// TwinCAT 3 PLC project Motor_test
// ProgramVersion: 3.1.4023.0
// libraries:
//   Tc2_ControllerToolbox, * (Beckhoff Automation GmbH)
//   Tc2_MC2, * (Beckhoff Automation GmbH)
//   Tc2_NCI, * (Beckhoff Automation GmbH)
//   Tc2_NcKinematicTransformation, * (Beckhoff Automation GmbH)
//   Tc2_PlcInterpolation, * (Beckhoff Automation GmbH)
//   Tc2_Standard, * (Beckhoff Automation GmbH)
//   Tc2_System, * (Beckhoff Automation GmbH)
//   Tc3_Module, * (Beckhoff Automation GmbH)
//   VisuSymbols,3.5.10.0,System
// project tree:
//   / GlobalTextList.TcGTLO, PlcTask.TcTTO, Visualization Manager.TcVMO (not stored)
//   POUs/ FB_CheckCurrentState.TcPOU, FB_ExecuteGcode.TcPOU, FB_GetPrinterParameters.TcPOU, FB_GetTemperature.TcPOU, FB_PowerChannel.TcPOU, FB_SteinhartEquation.TcPOU, Heater_control.TcPOU, MAIN.TcPOU, FB_PWM.TcPOU
//   VISUs/ Visualization.TcVIS
// real-time tasks:
//   TASK PlcTask: cycle T#1ms, priority 20, ADS port 350
// motion (NC):
//   TASK NC-Task 1 SAF: cycle T#1ms, priority 4, ADS port 501
//   TASK NC-Task 1 SVB: cycle T#1ms, priority 8, ADS port 511
//   AXIS axis xy 1 (id 1)
//     Dynamic: AccelerationMaximum=2000, DecelerationMaximum=2000, Acceleration=1000, Deceleration=1000
//     Velo: SlowManual=50, FastManual=100, Maximum=500
//     OtherSettings: AllowMotionCmdToSlave=true
//     encoder EncType=4
//       EncPara: ScaleFactorNumerator=40, ScaleFactorDenominator=12800, MaxCount=#x0000ffff
//         Inc: RefSoftSyncMask=#x0000ffff
//     drive DrvType=24
//       Analog: VeloReferenz=400, TorqueSetpointScale=10, ScaleFactorActTorque=0.1
//       TimeComp: TaskDelayCycles=1
//     controller CtrType=1
//       CtrPara: PriorControlFactor=1
//         Observer: BandWidth=20
//   AXIS axis xy 2 (id 2)
//     Dynamic: AccelerationMaximum=2000, DecelerationMaximum=2000, Acceleration=1000, Deceleration=1000
//     Velo: SlowManual=50, FastManual=100, Maximum=500
//     OtherSettings: AllowMotionCmdToSlave=true
//     encoder EncType=4
//       EncPara: ScaleFactorNumerator=40, ScaleFactorDenominator=12800, MaxCount=#x0000ffff
//         Inc: RefSoftSyncMask=#x0000ffff
//     drive DrvType=24
//       Analog: VeloReferenz=400, TorqueSetpointScale=10, ScaleFactorActTorque=0.1
//       TimeComp: TaskDelayCycles=1
//     controller CtrType=1
//       CtrPara: PriorControlFactor=1
//         Observer: BandWidth=20
//   AXIS Z axis (id 3)
//     Dynamic: AccelerationMaximum=100, DecelerationMaximum=100, Acceleration=50, Deceleration=50, Jerk=1000
//     Velo: RefSearch=3, RefSync=3, SlowManual=1, FastManual=4, Maximum=10
//     OtherSettings: AllowMotionCmdToSlave=true
//     encoder EncType=4
//       EncPara: ScaleFactorNumerator=8, ScaleFactorDenominator=12800, MaxCount=#x0000ffff
//         SoftEndMaxControl: Range=400
//         Inc: RefSearchInverse=true, RefSyncInverse=false, RefPosition=0.4, RefMode=1, RefSoftSyncMask=#x0000ffff
//     drive DrvType=24
//       Analog: VeloReferenz=80, TorqueSetpointScale=10, ScaleFactorActTorque=0.1
//       TimeComp: TaskDelayCycles=1
//     controller CtrType=1
//       CtrPara: PriorControlFactor=1
//         Observer: BandWidth=20
//   AXIS Extruder (id 4)
//     Dynamic: AccelerationMaximum=400, DecelerationMaximum=400, Acceleration=200, Deceleration=200, Jerk=500
//     Velo: SlowManual=1, FastManual=2, Maximum=100
//     OtherSettings: AllowMotionCmdToSlave=true
//     encoder EncType=4
//       EncPara: ScaleFactorNumerator=22.857, ScaleFactorDenominator=12800, MaxCount=#x0000ffff
//         Inc: RefSoftSyncMask=#x0000ffff
//     drive DrvType=24
//       Analog: VeloReferenz=50, TorqueSetpointScale=10, ScaleFactorActTorque=0.1
//       TimeComp: TaskDelayCycles=1
//     controller CtrType=1
//       CtrPara: PriorControlFactor=1
//         PosDiffControl: Range=15
//         Observer: BandWidth=20
//   AXIS X axis (id 5)
//     Dynamic: AccelerationMaximum=2000, DecelerationMaximum=2000, Acceleration=1000, Deceleration=1000
//     Velo: RefSearch=20, RefSync=20, SlowManual=20, FastManual=40, Maximum=500
//     OtherSettings: AllowMotionCmdToSlave=true
//     encoder EncType=1
//       EncPara: ScaleFactorNumerator=1, ScaleFactorDenominator=0.1
//         SoftEndMaxControl: Range=300
//     drive DrvType=5
//       Analog: VeloReferenz=500, TorqueSetpointScale=10, ScaleFactorActTorque=0.1
//       TimeComp: TaskDelayCycles=1
//     controller CtrType=1
//       CtrPara: PriorControlFactor=1
//         Observer: BandWidth=20
//   AXIS Y axis (id 6)
//     Dynamic: AccelerationMaximum=2000, DecelerationMaximum=2000, Acceleration=1000, Deceleration=1000
//     Velo: RefSearch=15, RefSync=15, SlowManual=15, FastManual=40, Maximum=500
//     OtherSettings: AllowMotionCmdToSlave=true
//     encoder EncType=1
//       SoftEndMaxControl: Range=300
//     drive DrvType=5
//       Analog: VeloReferenz=500, TorqueSetpointScale=10, ScaleFactorActTorque=0.1
//       TimeComp: TaskDelayCycles=1
//     controller CtrType=1
//       CtrPara: PriorControlFactor=1
//         Observer: BandWidth=20
// I/O:
//   DEVICE Device 3 (EtherCAT), AmsNetId 5.68.190.166.4.1
//     Term 1 (EK1101) [EK1101 EtherCAT Coupler (2A E-Bus, ID switch)]
//       Term 2 (EL9227-5500) [EL9227-5500 Overcurrent protection 24V DC, 2Ch., max. 10A (sum), adjustable, extended functionalities]
//       Term 3 (EL2024) [EL2024 4Ch. Dig. Output 24V, 2A]
//       Term 15 (EL3204-0200) [EL3204-0200 4Ch. Ana. In. PT1000 (RTD)]
//       Term 5 (EL1004) [EL1004 4Ch. Dig. Input 24V, 3ms]
//       Term 6 (EL7037) [EL7037 1Ch. Stepper motor output stage (24V, 1.5A)]
//       Term 7 (EL7037) [EL7037 1Ch. Stepper motor output stage (24V, 1.5A)]
//       Term 8 (EL7037) [EL7037 1Ch. Stepper motor output stage (24V, 1.5A)]
//       Term 9 (EL7037) [EL7037 1Ch. Stepper motor output stage (24V, 1.5A)]
//       Term 10 (EL9227-5500) [EL9227-5500 Overcurrent protection 24V DC, 2Ch., max. 10A (sum), adjustable, extended functionalities]
//       Term 11 (EL9011) [EL9011 End Terminal]
// variable links:
//   NC-Task 1 SAF/Axes/Extruder <-> Device 3 (EtherCAT)/Term 1 (EK1101)/Term 9 (EL7037)
//     Drive/Inputs/In/nState1 @bit 3 <-> STM Status/Status/Error
//     Drive/Inputs/In/nState1 @bit 7 <-> STM Status/Status/Motor stall
//     Drive/Inputs/In/nState1 @bit 5 <-> STM Status/Status/Moving negative
//     Drive/Inputs/In/nState1 @bit 4 <-> STM Status/Status/Moving positive
//     Drive/Inputs/In/nState1 @bit 1 <-> STM Status/Status/Ready
//     Drive/Inputs/In/nState1 <-> STM Status/Status/Ready to enable
//     Drive/Inputs/In/nState1 @bit 6 <-> STM Status/Status/Torque reduced
//     Drive/Inputs/In/nState1 @bit 2 <-> STM Status/Status/Warning
//     Drive/Inputs/In/nState2 @bit 3 <-> STM Status/Status/Digital input 1
//     Drive/Inputs/In/nState2 @bit 4 <-> STM Status/Status/Digital input 2
//     Drive/Inputs/In/nState2 @bit 5 <-> STM Status/Status/Sync error
//     Drive/Inputs/In/nState2 @bit 7 <-> STM Status/Status/TxPDO Toggle
//     Drive/Inputs/In/nState4 @bit 1 <-> WcState/InputToggle
//     Drive/Inputs/In/nState4 <-> WcState/WcState
//     Drive/Outputs/Out/nCtrl1 <-> STM Control/Control/Enable
//     Drive/Outputs/Out/nCtrl1 @bit 2 <-> STM Control/Control/Reduce torque
//     Drive/Outputs/Out/nCtrl1 @bit 1 <-> STM Control/Control/Reset
//     Drive/Outputs/Out/nCtrl2 @bit 3 <-> STM Control/Control/Digital output 1
//     Drive/Outputs/Out/nDataOut2[0] <-> STM Velocity/Velocity
//     Enc/Inputs/In/nDataIn1[0] <-> ENC Status compact/Counter value
//     Enc/Inputs/In/nDataIn2[0] <-> ENC Status compact/Latch value
//     Enc/Inputs/In/nState1 @bit 4 <-> ENC Status compact/Status/Counter overflow
//     Enc/Inputs/In/nState1 @bit 3 <-> ENC Status compact/Status/Counter underflow
//     Enc/Inputs/In/nState1 @bit 7 <-> ENC Status compact/Status/Extrapolation stall
//     Enc/Inputs/In/nState1 <-> ENC Status compact/Status/Latch C valid
//     Enc/Inputs/In/nState1 @bit 1 <-> ENC Status compact/Status/Latch extern valid
//     Enc/Inputs/In/nState1 @bit 2 <-> ENC Status compact/Status/Set counter done
//     Enc/Inputs/In/nState2 @bit 4 <-> ENC Status compact/Status/Status of extern latch
//     Enc/Inputs/In/nState2 <-> ENC Status compact/Status/Status of input A
//     Enc/Inputs/In/nState2 @bit 1 <-> ENC Status compact/Status/Status of input B
//     Enc/Inputs/In/nState2 @bit 2 <-> ENC Status compact/Status/Status of input C
//     Enc/Inputs/In/nState2 @bit 5 <-> ENC Status compact/Status/Sync error
//     Enc/Inputs/In/nState2 @bit 7 <-> ENC Status compact/Status/TxPDO Toggle
//     Enc/Inputs/In/nState4 @bit 1 <-> WcState/InputToggle
//     Enc/Inputs/In/nState4 <-> WcState/WcState
//     Enc/Outputs/Out/nCtrl1 <-> ENC Control compact/Control/Enable latch C
//     Enc/Outputs/Out/nCtrl1 @bit 3 <-> ENC Control compact/Control/Enable latch extern on negative edge
//     Enc/Outputs/Out/nCtrl1 @bit 1 <-> ENC Control compact/Control/Enable latch extern on positive edge
//     Enc/Outputs/Out/nCtrl1 @bit 2 <-> ENC Control compact/Control/Set counter
//     Enc/Outputs/Out/nDataOut1[0] <-> ENC Control compact/Set counter value
//   NC-Task 1 SAF/Axes/Z axis <-> Device 3 (EtherCAT)/Term 1 (EK1101)/Term 8 (EL7037)
//     Drive/Inputs/In/nState1 @bit 3 <-> STM Status/Status/Error
//     Drive/Inputs/In/nState1 @bit 7 <-> STM Status/Status/Motor stall
//     Drive/Inputs/In/nState1 @bit 5 <-> STM Status/Status/Moving negative
//     Drive/Inputs/In/nState1 @bit 4 <-> STM Status/Status/Moving positive
//     Drive/Inputs/In/nState1 @bit 1 <-> STM Status/Status/Ready
//     Drive/Inputs/In/nState1 <-> STM Status/Status/Ready to enable
//     Drive/Inputs/In/nState1 @bit 6 <-> STM Status/Status/Torque reduced
//     Drive/Inputs/In/nState1 @bit 2 <-> STM Status/Status/Warning
//     Drive/Inputs/In/nState2 @bit 3 <-> STM Status/Status/Digital input 1
//     Drive/Inputs/In/nState2 @bit 4 <-> STM Status/Status/Digital input 2
//     Drive/Inputs/In/nState2 @bit 5 <-> STM Status/Status/Sync error
//     Drive/Inputs/In/nState2 @bit 7 <-> STM Status/Status/TxPDO Toggle
//     Drive/Inputs/In/nState4 @bit 1 <-> WcState/InputToggle
//     Drive/Inputs/In/nState4 <-> WcState/WcState
//     Drive/Outputs/Out/nCtrl1 <-> STM Control/Control/Enable
//     Drive/Outputs/Out/nCtrl1 @bit 2 <-> STM Control/Control/Reduce torque
//     Drive/Outputs/Out/nCtrl1 @bit 1 <-> STM Control/Control/Reset
//     Drive/Outputs/Out/nCtrl2 @bit 3 <-> STM Control/Control/Digital output 1
//     Drive/Outputs/Out/nDataOut2[0] <-> STM Velocity/Velocity
//     Enc/Inputs/In/nDataIn1[0] <-> ENC Status compact/Counter value
//     Enc/Inputs/In/nDataIn2[0] <-> ENC Status compact/Latch value
//     Enc/Inputs/In/nState1 @bit 4 <-> ENC Status compact/Status/Counter overflow
//     Enc/Inputs/In/nState1 @bit 3 <-> ENC Status compact/Status/Counter underflow
//     Enc/Inputs/In/nState1 @bit 7 <-> ENC Status compact/Status/Extrapolation stall
//     Enc/Inputs/In/nState1 <-> ENC Status compact/Status/Latch C valid
//     Enc/Inputs/In/nState1 @bit 1 <-> ENC Status compact/Status/Latch extern valid
//     Enc/Inputs/In/nState1 @bit 2 <-> ENC Status compact/Status/Set counter done
//     Enc/Inputs/In/nState2 @bit 4 <-> ENC Status compact/Status/Status of extern latch
//     Enc/Inputs/In/nState2 <-> ENC Status compact/Status/Status of input A
//     Enc/Inputs/In/nState2 @bit 1 <-> ENC Status compact/Status/Status of input B
//     Enc/Inputs/In/nState2 @bit 2 <-> ENC Status compact/Status/Status of input C
//     Enc/Inputs/In/nState2 @bit 5 <-> ENC Status compact/Status/Sync error
//     Enc/Inputs/In/nState2 @bit 7 <-> ENC Status compact/Status/TxPDO Toggle
//     Enc/Inputs/In/nState4 @bit 1 <-> WcState/InputToggle
//     Enc/Inputs/In/nState4 <-> WcState/WcState
//     Enc/Outputs/Out/nCtrl1 <-> ENC Control compact/Control/Enable latch C
//     Enc/Outputs/Out/nCtrl1 @bit 3 <-> ENC Control compact/Control/Enable latch extern on negative edge
//     Enc/Outputs/Out/nCtrl1 @bit 1 <-> ENC Control compact/Control/Enable latch extern on positive edge
//     Enc/Outputs/Out/nCtrl1 @bit 2 <-> ENC Control compact/Control/Set counter
//     Enc/Outputs/Out/nDataOut1[0] <-> ENC Control compact/Set counter value
//   NC-Task 1 SAF/Axes/axis xy 1 <-> Device 3 (EtherCAT)/Term 1 (EK1101)/Term 6 (EL7037)
//     Drive/Inputs/In/nState1 @bit 3 <-> STM Status/Status/Error
//     Drive/Inputs/In/nState1 @bit 7 <-> STM Status/Status/Motor stall
//     Drive/Inputs/In/nState1 @bit 5 <-> STM Status/Status/Moving negative
//     Drive/Inputs/In/nState1 @bit 4 <-> STM Status/Status/Moving positive
//     Drive/Inputs/In/nState1 @bit 1 <-> STM Status/Status/Ready
//     Drive/Inputs/In/nState1 <-> STM Status/Status/Ready to enable
//     Drive/Inputs/In/nState1 @bit 6 <-> STM Status/Status/Torque reduced
//     Drive/Inputs/In/nState1 @bit 2 <-> STM Status/Status/Warning
//     Drive/Inputs/In/nState2 @bit 3 <-> STM Status/Status/Digital input 1
//     Drive/Inputs/In/nState2 @bit 4 <-> STM Status/Status/Digital input 2
//     Drive/Inputs/In/nState2 @bit 5 <-> STM Status/Status/Sync error
//     Drive/Inputs/In/nState2 @bit 7 <-> STM Status/Status/TxPDO Toggle
//     Drive/Inputs/In/nState4 @bit 1 <-> WcState/InputToggle
//     Drive/Inputs/In/nState4 <-> WcState/WcState
//     Drive/Outputs/Out/nCtrl1 <-> STM Control/Control/Enable
//     Drive/Outputs/Out/nCtrl1 @bit 2 <-> STM Control/Control/Reduce torque
//     Drive/Outputs/Out/nCtrl1 @bit 1 <-> STM Control/Control/Reset
//     Drive/Outputs/Out/nCtrl2 @bit 3 <-> STM Control/Control/Digital output 1
//     Drive/Outputs/Out/nDataOut2[0] <-> STM Velocity/Velocity
//     Enc/Inputs/In/nDataIn1[0] <-> ENC Status compact/Counter value
//     Enc/Inputs/In/nDataIn2[0] <-> ENC Status compact/Latch value
//     Enc/Inputs/In/nState1 @bit 4 <-> ENC Status compact/Status/Counter overflow
//     Enc/Inputs/In/nState1 @bit 3 <-> ENC Status compact/Status/Counter underflow
//     Enc/Inputs/In/nState1 @bit 7 <-> ENC Status compact/Status/Extrapolation stall
//     Enc/Inputs/In/nState1 <-> ENC Status compact/Status/Latch C valid
//     Enc/Inputs/In/nState1 @bit 1 <-> ENC Status compact/Status/Latch extern valid
//     Enc/Inputs/In/nState1 @bit 2 <-> ENC Status compact/Status/Set counter done
//     Enc/Inputs/In/nState2 @bit 4 <-> ENC Status compact/Status/Status of extern latch
//     Enc/Inputs/In/nState2 <-> ENC Status compact/Status/Status of input A
//     Enc/Inputs/In/nState2 @bit 1 <-> ENC Status compact/Status/Status of input B
//     Enc/Inputs/In/nState2 @bit 2 <-> ENC Status compact/Status/Status of input C
//     Enc/Inputs/In/nState2 @bit 5 <-> ENC Status compact/Status/Sync error
//     Enc/Inputs/In/nState2 @bit 7 <-> ENC Status compact/Status/TxPDO Toggle
//     Enc/Inputs/In/nState4 @bit 1 <-> WcState/InputToggle
//     Enc/Inputs/In/nState4 <-> WcState/WcState
//     Enc/Outputs/Out/nCtrl1 <-> ENC Control compact/Control/Enable latch C
//     Enc/Outputs/Out/nCtrl1 @bit 3 <-> ENC Control compact/Control/Enable latch extern on negative edge
//     Enc/Outputs/Out/nCtrl1 @bit 1 <-> ENC Control compact/Control/Enable latch extern on positive edge
//     Enc/Outputs/Out/nCtrl1 @bit 2 <-> ENC Control compact/Control/Set counter
//     Enc/Outputs/Out/nDataOut1[0] <-> ENC Control compact/Set counter value
//   NC-Task 1 SAF/Axes/axis xy 2 <-> Device 3 (EtherCAT)/Term 1 (EK1101)/Term 7 (EL7037)
//     Drive/Inputs/In/nState1 @bit 3 <-> STM Status/Status/Error
//     Drive/Inputs/In/nState1 @bit 7 <-> STM Status/Status/Motor stall
//     Drive/Inputs/In/nState1 @bit 5 <-> STM Status/Status/Moving negative
//     Drive/Inputs/In/nState1 @bit 4 <-> STM Status/Status/Moving positive
//     Drive/Inputs/In/nState1 @bit 1 <-> STM Status/Status/Ready
//     Drive/Inputs/In/nState1 <-> STM Status/Status/Ready to enable
//     Drive/Inputs/In/nState1 @bit 6 <-> STM Status/Status/Torque reduced
//     Drive/Inputs/In/nState1 @bit 2 <-> STM Status/Status/Warning
//     Drive/Inputs/In/nState2 @bit 3 <-> STM Status/Status/Digital input 1
//     Drive/Inputs/In/nState2 @bit 4 <-> STM Status/Status/Digital input 2
//     Drive/Inputs/In/nState2 @bit 5 <-> STM Status/Status/Sync error
//     Drive/Inputs/In/nState2 @bit 7 <-> STM Status/Status/TxPDO Toggle
//     Drive/Inputs/In/nState4 @bit 1 <-> WcState/InputToggle
//     Drive/Inputs/In/nState4 <-> WcState/WcState
//     Drive/Outputs/Out/nCtrl1 <-> STM Control/Control/Enable
//     Drive/Outputs/Out/nCtrl1 @bit 2 <-> STM Control/Control/Reduce torque
//     Drive/Outputs/Out/nCtrl1 @bit 1 <-> STM Control/Control/Reset
//     Drive/Outputs/Out/nCtrl2 @bit 3 <-> STM Control/Control/Digital output 1
//     Drive/Outputs/Out/nDataOut2[0] <-> STM Velocity/Velocity
//     Enc/Inputs/In/nDataIn1[0] <-> ENC Status compact/Counter value
//     Enc/Inputs/In/nDataIn2[0] <-> ENC Status compact/Latch value
//     Enc/Inputs/In/nState1 @bit 4 <-> ENC Status compact/Status/Counter overflow
//     Enc/Inputs/In/nState1 @bit 3 <-> ENC Status compact/Status/Counter underflow
//     Enc/Inputs/In/nState1 @bit 7 <-> ENC Status compact/Status/Extrapolation stall
//     Enc/Inputs/In/nState1 <-> ENC Status compact/Status/Latch C valid
//     Enc/Inputs/In/nState1 @bit 1 <-> ENC Status compact/Status/Latch extern valid
//     Enc/Inputs/In/nState1 @bit 2 <-> ENC Status compact/Status/Set counter done
//     Enc/Inputs/In/nState2 @bit 4 <-> ENC Status compact/Status/Status of extern latch
//     Enc/Inputs/In/nState2 <-> ENC Status compact/Status/Status of input A
//     Enc/Inputs/In/nState2 @bit 1 <-> ENC Status compact/Status/Status of input B
//     Enc/Inputs/In/nState2 @bit 2 <-> ENC Status compact/Status/Status of input C
//     Enc/Inputs/In/nState2 @bit 5 <-> ENC Status compact/Status/Sync error
//     Enc/Inputs/In/nState2 @bit 7 <-> ENC Status compact/Status/TxPDO Toggle
//     Enc/Inputs/In/nState4 @bit 1 <-> WcState/InputToggle
//     Enc/Inputs/In/nState4 <-> WcState/WcState
//     Enc/Outputs/Out/nCtrl1 <-> ENC Control compact/Control/Enable latch C
//     Enc/Outputs/Out/nCtrl1 @bit 3 <-> ENC Control compact/Control/Enable latch extern on negative edge
//     Enc/Outputs/Out/nCtrl1 @bit 1 <-> ENC Control compact/Control/Enable latch extern on positive edge
//     Enc/Outputs/Out/nCtrl1 @bit 2 <-> ENC Control compact/Control/Set counter
//     Enc/Outputs/Out/nDataOut1[0] <-> ENC Control compact/Set counter value
//   Motor test/Motor test Instance <-> Device 3 (EtherCAT)/Term 1 (EK1101)/Term 15 (EL3204-0200)
//     PlcTask Inputs/MAIN.hotbedResitance <-> RTD Inputs Channel 2/Value
//     PlcTask Inputs/MAIN.hotendResitance <-> RTD Inputs Channel 1/Value
//   Motor test/Motor test Instance <-> Device 3 (EtherCAT)/Term 1 (EK1101)/Term 3 (EL2024)
//     PlcTask Outputs/MAIN.hotbedHeater <-> Channel 4/Output
//     PlcTask Outputs/MAIN.hotendFan1 <-> Channel 1/Output
//     PlcTask Outputs/MAIN.hotendFan2 <-> Channel 2/Output
//     PlcTask Outputs/MAIN.hotendHeater <-> Channel 3/Output
//   Motor test/Motor test Instance <-> Device 3 (EtherCAT)/Term 1 (EK1101)/Term 5 (EL1004)
//     PlcTask Inputs/MAIN.HomingSensorX <-> Channel 2/Input
//     PlcTask Inputs/MAIN.HomingSensorY <-> Channel 1/Input
//     PlcTask Inputs/MAIN.HomingSensorZ <-> Channel 4/Input
//   Motor test/Motor test Instance <-> NC-Task 1 SAF/Axes/Extruder
//     PlcTask Inputs/MAIN.Extruder.NcToPlc <-> Outputs/ToPlc
//     PlcTask Outputs/MAIN.Extruder.PlcToNc <-> Inputs/FromPlc
//   Motor test/Motor test Instance <-> NC-Task 1 SAF/Axes/X axis
//     PlcTask Inputs/MAIN.Xaxis.NcToPlc <-> Outputs/ToPlc
//     PlcTask Outputs/MAIN.Xaxis.PlcToNc <-> Inputs/FromPlc
//   Motor test/Motor test Instance <-> NC-Task 1 SAF/Axes/Y axis
//     PlcTask Inputs/MAIN.Yaxis.NcToPlc <-> Outputs/ToPlc
//     PlcTask Outputs/MAIN.Yaxis.PlcToNc <-> Inputs/FromPlc
//   Motor test/Motor test Instance <-> NC-Task 1 SAF/Axes/Z axis
//     PlcTask Inputs/MAIN.Zaxis.NcToPlc <-> Outputs/ToPlc
//     PlcTask Outputs/MAIN.Zaxis.PlcToNc <-> Inputs/FromPlc
//   Motor test/Motor test Instance <-> NC-Task 1 SAF/Axes/axis xy 1
//     PlcTask Inputs/MAIN.XY_1.NcToPlc <-> Outputs/ToPlc
//     PlcTask Outputs/MAIN.XY_1.PlcToNc <-> Inputs/FromPlc
//   Motor test/Motor test Instance <-> NC-Task 1 SAF/Axes/axis xy 2
//     PlcTask Inputs/MAIN.XY_2.NcToPlc <-> Outputs/ToPlc
//     PlcTask Outputs/MAIN.XY_2.PlcToNc <-> Inputs/FromPlc
//   Motor test/Motor test Instance <-> NC-Task 1 SAF/NCI XYZ
//     PlcTask Inputs/MAIN.in_stNciToPlc <-> Outputs/ToPlc
//     PlcTask Outputs/MAIN.out_stPlcToNci <-> Inputs/FromPlc
//   Motor test/Motor test Instance <-> NC-Task 1 SAF/XY core
//     PlcTask Inputs/MAIN.in_stKinToPlc <-> Outputs/ToPlc

CONFIGURATION Motor_test
    RESOURCE PLC ON TwinCAT3
        TASK PlcTask(INTERVAL := T#1ms, PRIORITY := 20);
        PROGRAM MAIN WITH PlcTask : MAIN;
    END_RESOURCE
END_CONFIGURATION

// ---- POUs/MAIN.TcPOU
PROGRAM MAIN
VAR
	
	fbPower: FB_PowerChannel;
	
	//fbfanControl: Fan_control;
	fbHotEndHeatingControl: Heater_control;
	fbGetHotEndTemperature : FB_GetTemperature;
	fbHotBedHeatingControl: Heater_control;
	fbGetHotBedTemperature : FB_GetTemperature;
	fbGetCurrentState: FB_CheckCurrentState;
	fbGetPrinterParameters: FB_GetPrinterParameters;
	
	fbConfirmHsk: ItpConfirmHsk;
	fbExecuteGcode: FB_ExecuteGcode;
	fbBuildGroup: CfgBuildExt3DGroup;
	fbReconfigAxis: CfgReconfigAxis;
	fbAddAxis: CfgAddAxisToGroup;
	fbLoadGCode: ItpLoadProgEx;
	fbStartGCode: ItpStartStopEx;
	fbConfigKinGroup: FB_KinConfigGroup;
    stAxesConfig: ST_KinAxes;
	in_stKinToPlc AT %I*  : NCTOPLC_NCICHANNEL_REF;
	
	Xaxis: AXIS_REF;
	Yaxis: AXIS_REF;
	Zaxis: AXIS_REF;
	Extruder: AXIS_REF;
	XY_1: AXIS_REF;
	XY_2: AXIS_REF;

	setXY1:MC_SetPosition;
	setXY2:MC_SetPosition;
	setExtruder:MC_SetPosition;
	
	Zhome: MC_Home;
	
	Xjog: MC_Jog;
	Yjog: MC_Jog;
	moveExtruderAbsolute1: MC_MoveAbsolute;
	moveExtruderAbsolute2: MC_MoveAbsolute;
	moveZAbsolute: MC_MoveAbsolute;
	moveXAbsolute: MC_MoveAbsolute;
	moveYAbsolute: MC_MoveAbsolute;
	
	ExecuteKinConfig: BOOL := true;
	HomingSensorX AT %I*: BOOL;
	HomingSensorY AT %I*: BOOL;
	HomingSensorZ AT %I*: BOOL;
	
	
	in_stNciToPlc AT %I*: NCTOPLC_NCICHANNEL_REF;
	out_stPlcToNci AT %Q*: PLCTONC_NCICHANNEL_REF;
	
	Xoffset: LREAL := 0;
	Yoffset: LREAL := 0;
	Zoffset: LREAL := 0.38;
	

	hotendResitance AT %I*  : INT := 1;
	hotbedResitance AT %I*  : INT := 1;
	hotendHeater AT %Q*  : BOOL;
	hotbedHeater AT %Q*  : BOOL;
	hotendFan1 AT %Q*  : BOOL;
	hotendFan2 AT %Q*  : BOOL;
	HeatersOn: BOOL := FALSE;
	
	// Verschillende temperturen met hun weerstanden voor de steinhart equation
	// temperaturen die dichter bij de use case zitten vebeter de precisie van de gemeten temperatuur
	hotEndCalibrationValues  : ARRAY [1..6] OF LREAL := [200 ,552.99 ,210 ,456.11, 220, 378.95];
	hotBedCalibrationValues : ARRAY [1..6] OF LREAL := [50 ,35262 ,60 ,24136 ,70 ,16841 ]; 
	
	ExtruderValue: LREAL;
	
	State: INT ;
	ExtruderSpeed : LREAL;
	sPrgNameSegment: STRING(255) := 'beckhoff.nc';
	nInterpreterState: UDINT;
	
	bEnable: BOOL := FALSE;
	homeAxi: BOOL := FALSE;
	executeGcode: BOOL := FALSE;
	moveAbs1: BOOL := FALSE;
	moveAbs2: BOOL := FALSE;
	executeExtruderMovement :BOOL := TRUE;
	resetExtruder : BOOL :=FALSE;
	intreperterState : UDINT;
	
END_VAR

fbPower(
	bEnable:=bEnable, 
	fOvr:= 100.0, 
	stX:=Xaxis, 
	stY:=Yaxis, 
	stZ:=Zaxis,
	stXY_1:= XY_1,
	stXY_2:= XY_2,
	stExt:= Extruder,
	stPlcToNci:=out_stPlcToNci , 
	bAllAxesReady=> );
	
moveExtruderAbsolute1(Axis := Extruder, execute := moveAbs1 , Position := extruderValue ,Velocity := extruderSpeed ,buffermode := MC_Aborting );
moveExtruderAbsolute2(Axis := Extruder, execute := moveAbs2 , Position := extruderValue ,Velocity := extruderSpeed ,buffermode := MC_Aborting );		
	
IF HeatersOn THEN	
	fbHotEndHeatingControl(terminalResistance := hotendResitance,desiredTemp := 60,calibrationValues := hotEndCalibrationValues, maxTemp := 220); // pd controlller die een pwm signaal output
	hotendHeater := fbHotEndHeatingControl.PWM_out;
	fbHotBedHeatingControl(terminalResistance := hotbedResitance,desiredTemp := 60,calibrationValues := hotBedCalibrationValues, maxTemp := 70); // pd controlller die een pwm signaal output
	hotbedHeater := fbHotBedHeatingControl.PWM_out;
ELSE 
	hotendHeater := FALSE;
	hotbedHeater := FALSE;
END_IF 
	
CASE State OF
	0: // init
	
	
	hotendFan1 := TRUE;
	hotendFan2 := TRUE;
	moveAbs1 := FALSE;
	moveAbs2 := FALSE;
	
	ExecuteKinConfig:=TRUE;
	IF fbPower.bAllAxesReady THEN
		State := 10; 
	END_IF
	
	
	
	10:
	HeatersOn:= TRUE;
	
	stAxesConfig.nAxisIdsAcs[1] := XY_2.NcToPlc.AxisId;
	stAxesConfig.nAxisIdsAcs[2] := XY_1.NcToPlc.AxisId;
	stAxesConfig.nAxisIdsMcs[1] := Xaxis.NcToPlc.AxisId;
	stAxesConfig.nAxisIdsMcs[2] := Yaxis.NcToPlc.AxisId;
	
	fbConfigKinGroup( // voeg de xy core motoren toe tot de kinematische groep
    bExecute       := ExecuteKinConfig ,
    bCartesianMode := TRUE ,
    stAxesList     := stAxesConfig,
    stKinRefIn     := in_stKinToPlc );
	
	IF NOT fbConfigKinGroup.bBusy THEN
		IF NOT fbConfigKinGroup.bError THEN
			ExecuteKinConfig:=FALSE;
			fbConfigKinGroup(
			bExecute       := ExecuteKinConfig ,
			stAxesList     := stAxesConfig,
			stKinRefIn     := in_stKinToPlc );
			IF homeAxi THEN
				State:=20;
			END_IF
		END_IF
	ELSIF F_KinGetChnOperationState(in_stKinToPlc) = KinStatus_Ready THEN
		ExecuteKinConfig:=FALSE;
			fbConfigKinGroup(
			bExecute       := ExecuteKinConfig ,
			stAxesList     := stAxesConfig,
			stKinRefIn     := in_stKinToPlc );
			IF homeAxi THEN
				State:=20;
			END_IF
	END_IF
	
	
	
	20: // jog de x axis tot de eind switch wordt geraakt
	Xjog(Axis:= Xaxis,JogBackwards:= TRUE , Deceleration:= 1500);
	
	IF NOT HomingSensorX THEN
		Xjog(Axis:= Xaxis,JogBackwards:= FALSE,);
		State:=21;
	END_IF
	
	
	
	21: // jog de y axis tot de eind switch wordt geraakt
	Yjog(Axis:= Yaxis,JogBackwards:= TRUE , Deceleration:= 1500);
	IF NOT HomingSensorY THEN
		Yjog(Axis:= Yaxis,JogBackwards:= FALSE);	
		State:=22;
	END_IF
	
	
	
	22: // Zet cartesian mode uit zodat de positie van de xy motoren op 0 geet kan worden om te homen
	ExecuteKinConfig:=TRUE;
	fbConfigKinGroup( 
    bExecute       := ExecuteKinConfig,
    bCartesianMode := FALSE ,
    stAxesList     := stAxesConfig,
    stKinRefIn     := in_stKinToPlc );
	
	
	IF NOT fbConfigKinGroup.bBusy THEN
		SetXY1(execute:= TRUE ,axis:= XY_1 ,position:= Xoffset);
		SetXY2(execute:= TRUE ,axis:= XY_2 ,position:= Yoffset);
		IF NOT fbConfigKinGroup.bError THEN
			ExecuteKinConfig:=FALSE;
			fbConfigKinGroup(
			bExecute       := ExecuteKinConfig ,
			stAxesList     := stAxesConfig,
			stKinRefIn     := in_stKinToPlc );
			State:=23;
		END_IF
	END_IF
	
	
	
	23: // home de z axis
	Zhome(axis := Zaxis,execute := TRUE,BCalibrationCam := NOT HomingSensorZ,Position := Zoffset);
	IF Zhome.Done THEN
		ExecuteKinConfig:=TRUE;
		State:=24;
	END_IF
	
	
	
	24:
	
	fbConfigKinGroup( // zet de kinematische groep weer op cartesian mode om hem weer te kunnnen bewegen.
    bExecute       := ExecuteKinConfig,
    bCartesianMode := TRUE ,
    stAxesList     := stAxesConfig,
    stKinRefIn     := in_stKinToPlc );
	
	IF NOT fbConfigKinGroup.bBusy THEN
		IF NOT fbConfigKinGroup.bError THEN
			State:= 25;
		END_IF
	END_IF
	
	
	25:
	moveZAbsolute(axis:= Zaxis, Execute:= TRUE, Position:= 1, velocity:=1);
	IF moveZAbsolute.Done THEN
		moveZAbsolute(axis:= Zaxis, Execute:= FALSE);
		state:= 26;
	END_IF
	
	
	26:
	setExtruder(execute:= TRUE ,axis:= Extruder ,position:= 0);
	IF setExtruder.Done AND fbGetHotEndTemperature.temperatureSensor >= 210 AND fbGetHotBedTemperature.temperatureSensor >= 55 THEN
		state:= 30;
	END_IF
	
	
	
	30: // het configureren van de NCI met de x,y en z as
	fbBuildGroup(
		bExecute:=TRUE,
		nGroupId:=ItpGetGroupId(sNciToPlc:=in_stNciToPlc),
		nXAxisId:=XAxis.NcToPlc.AxisId,
		nYAxisId:=YAxis.NcToPlc.AxisId,
		nZAxisId:=ZAxis.NcToPlc.AxisId,
		tTimeOut:=T#2S );
		
	IF NOT fbBuildGroup.bBusy THEN
		fbBuildGroup( bExecute:=FALSE );
		
		IF NOT fbBuildGroup.bErr THEN
				State	:= 31;
		END_IF
	END_IF
	
	31:
	IF executeGcode THEN
		state:= 40;
	END_IF
	
	40: // laad segment 1
	fbExecuteGcode(execute:= TRUE ,sPrgName:= sPrgNameSegment ,in_stNciToPlc:= in_stNciToPlc, reset:= FALSE);
	
	IF fbExecuteGcode.done THEN
		fbExecuteGcode(execute:= FALSE, reset:= TRUE);
		state:= 41;
	END_IF
	
	
	
	41: //tijdens g-code 
	fbGetPrinterParameters(in_stNciToPlc:= in_stNciToPlc, extruderValue=> extruderValue,extruderSpeed=> extruderSpeed);
	fbGetCurrentState(in_stNciToPlc:= in_stNciToPlc, nextState:= 42, state=> State);
	
	moveAbs1 := TRUE;
	moveAbs2 := FALSE;
	42: //tijdens g-code absoluut commando 2
	fbGetPrinterParameters(in_stNciToPlc:= in_stNciToPlc, extruderValue=> extruderValue,extruderSpeed=> extruderSpeed);
	fbGetCurrentState(in_stNciToPlc:= in_stNciToPlc, nextState:= 42, state=> State);
	
	moveAbs1 := FALSE;
	moveAbs2 := TRUE;
	43: // set position extruder axis
	moveAbs1 := FALSE;
	moveAbs2 := FALSE;
	
	setExtruder(execute:= TRUE ,axis:= Extruder ,position:= 0);
	IF setExtruder.Done THEN
		fbConfirmHsk(sNciToPlc := in_stNciToPlc,
						  sPlcToNci:= out_stPlcToNci,
						  bExecute:= TRUE);
		setExtruder(execute:= FALSE ,axis:= Extruder);
	
		state:= 41;
	END_IF
	fbConfirmHsk(sNciToPlc := in_stNciToPlc,
						  sPlcToNci:= out_stPlcToNci,
						  bExecute:= FALSE);
						  
	50: // print is klaar
	moveXAbsolute(axis:= Xaxis, Execute:= TRUE, Position:= 10, velocity:=25);
	moveYAbsolute(axis:= Yaxis, Execute:= TRUE, Position:= 10, velocity:=25);
	IF moveXAbsolute.Done AND moveYAbsolute.Done THEN
		moveXAbsolute(axis:= Xaxis, Execute:= FALSE);
		moveYAbsolute(axis:= Yaxis, Execute:= FALSE);
		state:= 51;
	END_IF
	51: // doe niks
	HeatersOn:= FALSE;
	60:// rotzooi
	
	
END_CASE

END_PROGRAM

// ---- POUs/FB_PowerChannel.TcPOU
FUNCTION_BLOCK FB_PowerChannel
VAR_INPUT
	bEnable			: BOOL := FALSE;
	fOvr			: LREAL;
END_VAR
VAR_IN_OUT
	stX				: AXIS_REF;
	stY 			: AXIS_REF;
	stZ				: AXIS_REF;
	stXY_1			: AXIS_REF;
	stXY_2			: AXIS_REF;
	stExt			: AXIS_REF;
	stPlcToNci		: PLCTONC_NCICHANNEL_REF;
END_VAR
VAR_OUTPUT
	bAllAxesReady	: BOOL := FALSE;
END_VAR
VAR
	fbPowerX		:	MC_Power;
	fbPowerY		:	MC_Power;
	fbPowerZ		:	MC_Power;
	fbPowerXY_1		:	MC_Power;
	fbPowerXY_2		:	MC_Power;
	fbPowerExt		:	MC_Power;
END_VAR

fbPowerX( 
	Axis:=stX , 
	Enable:=bEnable , 
	Enable_Positive:= bEnable, 
	Enable_Negative:= bEnable, 
	Override:=fOvr , 
	BufferMode:= , 
	Status=> , 
	Busy=> , 
	Active=> , 
	Error=> , 
	ErrorID=> );
fbPowerY(
	Axis:=stY , 
	Enable:=bEnable , 
	Enable_Positive:= bEnable, 
	Enable_Negative:= bEnable, 
	Override:=fOvr , 
	BufferMode:= , 
	Status=> , 
	Busy=> , 
	Active=> , 
	Error=> , 
	ErrorID=> );
fbPowerZ(
	Axis:=stZ , 
	Enable:=bEnable , 
	Enable_Positive:= bEnable, 
	Enable_Negative:= bEnable, 
	Override:=fOvr , 
	BufferMode:= , 
	Status=> , 
	Busy=> , 
	Active=> , 
	Error=> , 
	ErrorID=> );
fbPowerXY_1(
	Axis:=stXY_1 , 
	Enable:=bEnable , 
	Enable_Positive:= bEnable, 
	Enable_Negative:= bEnable, 
	Override:=fOvr , 
	BufferMode:= , 
	Status=> , 
	Busy=> , 
	Active=> , 
	Error=> , 
	ErrorID=> );	
fbPowerXY_2(
	Axis:=stXY_2 , 
	Enable:=bEnable , 
	Enable_Positive:= bEnable, 
	Enable_Negative:= bEnable, 
	Override:=fOvr , 
	BufferMode:= , 
	Status=> , 
	Busy=> , 
	Active=> , 
	Error=> , 
	ErrorID=> );
fbPowerExt(
	Axis:=stExt, 
	Enable:=bEnable , 
	Enable_Positive:= bEnable, 
	Enable_Negative:= bEnable, 
	Override:=fOvr , 
	BufferMode:= , 
	Status=> , 
	Busy=> , 
	Active=> , 
	Error=> , 
	ErrorID=> );	
	
ItpSetOverridePercent(fOverridePercent:=fOvr, sPlcToNci:=stPlcToNci);

IF fbPowerX.Status AND fbPowerY.Status AND fbPowerZ.Status AND fbPowerXY_1.Status AND fbPowerXY_2.Status AND fbPowerExt.Status THEN
	bAllAxesReady	:= TRUE;
ELSE
	bAllAxesReady	:= FALSE;
END_IF

END_FUNCTION_BLOCK

// ---- POUs/Heater_control.TcPOU
FUNCTION_BLOCK Heater_control
VAR_INPUT
	terminalResistance: INT;
	desiredTemp: LREAL;
	calibrationValues: ARRAY [1..6] OF LREAL;
	maxTemp: LREAL;
END_VAR
VAR_OUTPUT
	PWM_out: BOOL;
END_VAR
VAR
	fbGetHotEndTemperature : FB_GetTemperature;
	
	realTemp: LREAL;
	temperature :LREAL;
	error: LREAL; // E(k)
	previousError: LREAL; // E(k-1)
	integral: LREAL;
	derivative: LREAL;
	cycleTime: LREAL;
	controlSignal: LREAL;
	PWM: FB_PWM;
	FB_GETCURTASKINDEX:GETCURTASKINDEX;
	PID : FB_CTRL_PID;
	
	PID_params : ST_CTRL_PID_PARAMS := ( tCtrlCycleTime := T#1MS,  tTaskCycleTime:= T#1MS,fKp := 40, tTn := T#1MS ,tTv := T#1MS,  tTd := T#1M );
	
	Kp : LREAL := 120;
	Ki : LREAL := 1.5;
	Kd : LREAL := 45;
	
END_VAR

IF fbGetHotEndTemperature.temperatureSensor < maxTemp THEN
	fbGetHotEndTemperature(terminalResistance := (10*INT_TO_REAL(terminalResistance)), calibrationValues := calibrationValues );// weerstand naar temperatuur conversie
	
	error := desiredTemp - fbGetHotEndTemperature.temperatureSensor;
	FB_GETCURTASKINDEX();
	cycleTime := (UDINT_TO_LREAL(_TaskInfo[FB_GETCURTASKINDEX.index].CycleTime)/ 10_000_000);
	//integral := integral + error * cycleTime;
	derivative := (error - previousError) / cycleTime;
	controlSignal := (Kp * error  + Kd * derivative); //+ Ki * integral
	
	
	IF (controlSignal > 0 ) THEN
		PWM( dutyCycle := controlSignal);	
	ELSE 
		PWM(dutyCycle := 0);
	END_IF
	
	PWM_out := PWM.state; 
	previousError := error;
ELSE 
	PWM_out := FALSE;
END_IF

END_FUNCTION_BLOCK

// ---- POUs/FB_GetTemperature.TcPOU
FUNCTION_BLOCK FB_GetTemperature
VAR_INPUT
	terminalResistance : LREAL := 1;
	
	//values based on the EPCOS B57560G104F NTS sensor
	calibrationValues : ARRAY [1..6] OF LREAL := [25 ,100000 ,100 ,6338.3 , 200, 552.99];
	
END_VAR
VAR_OUTPUT
	temperatureSensor : LREAL;
END_VAR
VAR
	FBSteinHart : FB_SteinhartEquation; 
	A : LREAL;
	B : LREAL;
	C : LREAL;
END_VAR

// vraag steinhart parameters op
FBSteinHart(CV := calibrationValues , A => A, B => B, C => C);
// temperatuur wordt berekent met steainhart parameters en vergelijking
temperatureSensor := 1/(A+ B*LN(terminalResistance) + C * EXPT(LN(terminalResistance),3)); // steinhart equation is used to calculate the temperature of the sensor

END_FUNCTION_BLOCK

// ---- POUs/FB_SteinhartEquation.TcPOU
FUNCTION_BLOCK FB_SteinhartEquation
VAR_INPUT
	CV : ARRAY [1..6] OF LREAL;
	
END_VAR
VAR_OUTPUT
	C: LREAL;
	B: LREAL;
	A: LREAL;
	
END_VAR
VAR
	L1: LREAL;
	L2: LREAL;
	L3: LREAL;
	
	Y1: LREAL;
	Y2: LREAL;
	Y3: LREAL;

	H1: LREAL;
	H2: LREAL;
	
END_VAR

 L1 := LN(CV[2]);
 L2 := LN(CV[4]);
 L3 := LN(CV[6]);
 
 Y1 := 1/CV[1];
 Y2 := 1/CV[3];
 Y3 := 1/CV[5];
   
 H1 := (Y2 - Y1)/(L2 - L1);
 H2 := (Y3 - Y1)/(L3 - L1);
 
 C := ((H2 - H1)/(L3 - L2))* EXPT((L1+L2+L3),-1);
 B := H1 - C*(EXPT(L1,2) + L1*L2 + EXPT(L2,2));
 A := Y1 - (B+EXPT(L1,2)*C)*L1;

END_FUNCTION_BLOCK

// ---- POUs/FB_PWM.TcPOU
FUNCTION_BLOCK FB_PWM
VAR_INPUT
	dutyCycle: LREAL;
END_VAR
VAR_OUTPUT
	state:BOOL;
END_VAR
VAR
	pulseWidth:LREAL := 0;
	hertz: LREAL;
	currentTimeStep:LREAL;
	FB_GETCURTASKINDEX:GETCURTASKINDEX;
END_VAR

// a simple PWM function
FB_GETCURTASKINDEX();
Hertz:= 1 / (UDINT_TO_LREAL(_TaskInfo[FB_GETCURTASKINDEX.index].CycleTime)/ 10_000_000); // function takes the cycle time of the system to calculate the hertz
currentTimeStep:= currentTimeStep+1;// go to the next step


IF currentTimeStep <= pulseWidth  AND currentTimeStep <= hertz THEN // time on
	state:=TRUE;
ELSIF currentTimeStep >= hertz THEN // when finished
	state:=FALSE;
	pulseWidth:= hertz * dutyCycle; // the value is onverted to in to get rid of the values after the dot
	currentTimeStep:=0;
ELSE // wehn pwm is off
	state := FALSE;
END_IF

END_FUNCTION_BLOCK

// ---- POUs/FB_CheckCurrentState.TcPOU
FUNCTION_block FB_CheckCurrentState
VAR_INPUT
	in_stNciToPlc: NCTOPLC_NCICHANNEL_REF;
	nextState: INT;
END_VAR
VAR_OUTPUT
	State: INT;
END_VAR
VAR
	nInterpreterState: UDINT;
END_VAR


nInterpreterState	:= ItpGetStateInterpreter(sNciToPlc:=in_stNciToPlc); // status van de NCI

IF ItpIsHskMFunc( in_stNciToPlc ) THEN // Bij m- function 1 gaan naar de set etruder position stte
	IF ItpGetHskMFunc( in_stNciToPlc ) = 1 THEN
		State:=43;
	END_IF
ELSIF nInterpreterState = Tc2_NCI.NCI_INTERPRETER_READY THEN
		State:=50;
	ELSE 
		state := nextState;
END_IF

END_FUNCTION_BLOCK

// ---- POUs/FB_GetPrinterParameters.TcPOU
FUNCTION_BLOCK FB_GetPrinterParameters
VAR_INPUT
	in_stNciToPlc: NCTOPLC_NCICHANNEL_REF;;
END_VAR
VAR_OUTPUT
	extruderValue: LREAL;
	extruderSpeed: LREAL;
END_VAR
VAR
	hParam: DINT;
	printerSpeed: LREAL;
END_VAR

hParam := ItpGetHParam( in_stNciToPlc );
extruderValue := (DINT_TO_LREAL (hParam)/100000);
printerSpeed := ItpGetSetPathVelocity( in_stNciToPlc );
extruderSpeed := (printerSpeed * 0.08);

IF extruderSpeed = 0  THEN // voorkomt dat de absolute commando een foutmeleding geeft
		extruderSpeed:= 0.01;
END_IF

END_FUNCTION_BLOCK

// ---- POUs/FB_ExecuteGcode.TcPOU
FUNCTION_BLOCK FB_ExecuteGcode
VAR_INPUT
	sPrgName: STRING(255);
	execute: BOOL;
	in_stNciToPlc: NCTOPLC_NCICHANNEL_REF;
	reset: bool := FALSE;
END_VAR
VAR_OUTPUT
	done: BOOL;
END_VAR
VAR
	state: INT := 0;
	nInterpreterState: UDINT;
	
	fbLoadGCode: ItpLoadProgEx;
	fbStartGCode: ItpStartStopEx;
	
END_VAR

CASE state OF
	0: // voer g-code uit 
	IF execute = TRUE THEN
		done:=FALSE;
		state:= 10;
	END_IF
	
	10:// laad g-code
	fbLoadGCode(
		sNciToPlc:=in_stNciToPlc, 
		bExecute:=TRUE, 
		sPrg:= sPrgName, 
		nLength:= INT_TO_UDINT(LEN(sPrgName)) );
	IF NOT fbLoadGCode.bBusy THEN
		IF NOT fbLoadGCode.bErr THEN
			State	:= 20;				
		END_IF
		fbLoadGCode(sNciToPlc:=in_stNciToPlc, bExecute:=FALSE); 
	END_IF 
	
	20:// check status NCI
	fbLoadGCode(
		sNciToPlc:=in_stNciToPlc, 
		bExecute:=FALSE);
	nInterpreterState	:= ItpGetStateInterpreter(sNciToPlc:=in_stNciToPlc);
	IF nInterpreterState = Tc2_NCI.NCI_INTERPRETER_READY THEN // als de interpreter klaar is kan het programma verder
			State	:= 30;	
	END_IF
	
	30: // start g-code
	fbStartGCode(
		bStart:=TRUE, 
		bStop:=FALSE, 
		tTimeOut:= , 
		sNciToPlc:= in_stNciToPlc, 
		bBusy=> , 
		bErr=> , 
		nErrId=> );
	IF NOT fbStartGCode.bBusy THEN
		IF NOT fbStartGCode.bErr THEN
			State	:= 40;			
		END_IF
		fbStartGCode( bStart:= FALSE, sNciToPlc:= in_stNciToPlc); 
	END_IF
	
	40: // g-code is gestart en functieblok is klaar
	fbStartGCode( bStart:= FALSE, sNciToPlc:= in_stNciToPlc);
	done := TRUE;
	state := 50;
	
	50: // reset functieblok
	IF reset = TRUE THEN
		state := 0;
	END_IF
	
END_CASE

END_FUNCTION_BLOCK

// ---- GlobalTextList.TcGTLO
TEXTLIST GlobalTextList
  48 = '%i'
  479 = 'Enable'
  715 = 'Execute'
  523 = 'Home'
  299 = 'Hot bed'
  980 = 'Hot End'
  21 = 'Hot end'
  948 = 'Hotbed'
  750 = 'Load gcode'
  49 = 'State'
  993 = 'Stop'
END_TEXTLIST

// ---- VISUs/Visualization.TcVIS
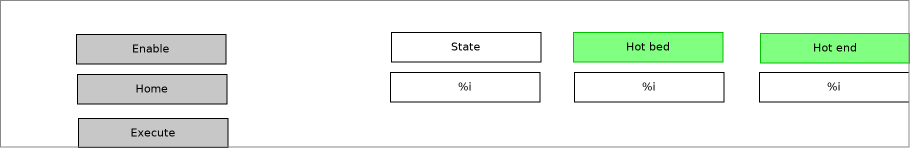
VISUALIZATION Visualization  // 910x148
    Rectangle (76,34 150x30), "Enable", colour toggle: MAIN.bEnable
        toggle MAIN.bEnable
    Rectangle (77,74 150x30), "Home", colour toggle: MAIN.homeAxi
        tap MAIN.homeAxi
    Rectangle (78,118 150x30), "Execute", colour toggle: MAIN.executeGcode
        tap MAIN.executeGcode
    Rectangle (390,72 150x30), "%i", text variable: MAIN.State
    Rectangle (391,32 150x30), "State"
    Rectangle (573,32 150x30), "Hot bed", colour toggle: MAIN.fbHotBedHeatingControl.TooHot
    Rectangle (759,72 150x30), "%i", text variable: MAIN.fbHotEndHeatingControl.temperatureSensor
    Rectangle (760,33 150x30), "Hot end", colour toggle: MAIN.fbHotEndHeatingControl.TooHot
    Rectangle (574,72 150x30), "%i", text variable: MAIN.fbHotBedHeatingControl.temperatureSensor
END_VISUALIZATION
